Omron CX-Programmer project NewProject (CX-Programmer 9.75)

# PLC NewPLC1: CP2E-N N

## Program NewProgram1 (cyclic task 0)

### Section Section1

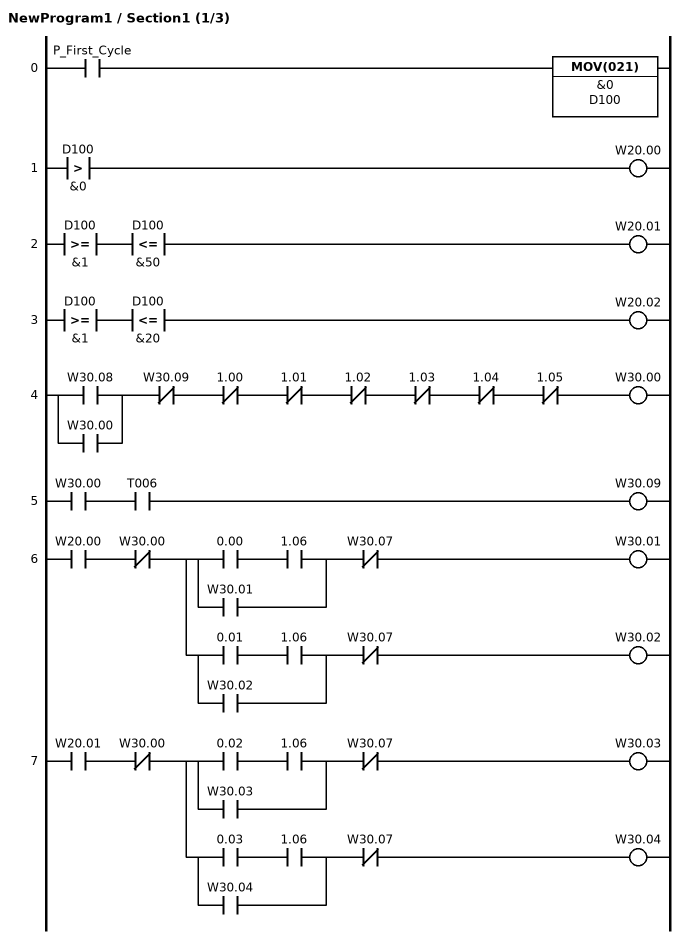
; rung 0
LD P_First_Cycle
MOV(021) &0 D100
; rung 1
LD>(320) D100 &0
OUT W20.00
; rung 2
LD>=(325) D100 &1
AND<=(315) D100 &50
OUT W20.01
; rung 3
LD>=(325) D100 &1
AND<=(315) D100 &20
OUT W20.02
; rung 4
LD W30.08
OR W30.00
ANDNOT W30.09
ANDNOT 1.00
ANDNOT 1.01
ANDNOT 1.02
ANDNOT 1.03
ANDNOT 1.04
ANDNOT 1.05
OUT W30.00
; rung 5
LD W30.00
AND T006
OUT W30.09
; rung 6
LD W20.00
ANDNOT W30.00
OUT TR0
LD 0.00
AND 1.06
OR W30.01
ANDLD
ANDNOT W30.07
OUT W30.01
LD TR0
LD 0.01
AND 1.06
OR W30.02
ANDLD
ANDNOT W30.07
OUT W30.02
; rung 7
LD W20.01
ANDNOT W30.00
OUT TR0
LD 0.02
AND 1.06
OR W30.03
ANDLD
ANDNOT W30.07
OUT W30.03
LD TR0
LD 0.03
AND 1.06
OR W30.04
ANDLD
ANDNOT W30.07
OUT W30.04

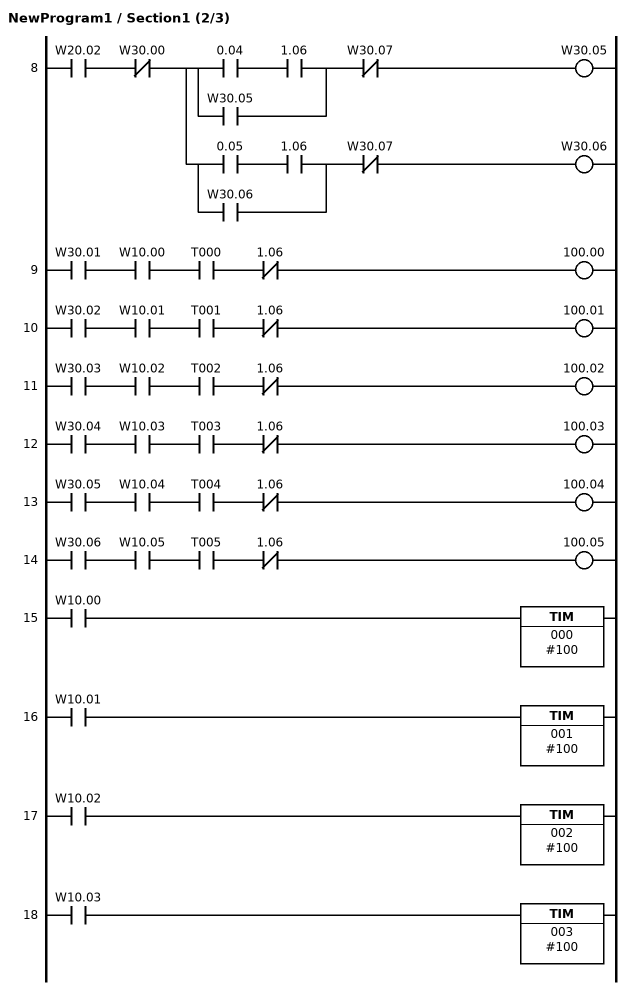
; rung 8
LD W20.02
ANDNOT W30.00
OUT TR0
LD 0.04
AND 1.06
OR W30.05
ANDLD
ANDNOT W30.07
OUT W30.05
LD TR0
LD 0.05
AND 1.06
OR W30.06
ANDLD
ANDNOT W30.07
OUT W30.06
; rung 9
LD W30.01
AND W10.00
AND T000
ANDNOT 1.06
OUT 100.00
; rung 10
LD W30.02
AND W10.01
AND T001
ANDNOT 1.06
OUT 100.01
; rung 11
LD W30.03
AND W10.02
AND T002
ANDNOT 1.06
OUT 100.02
; rung 12
LD W30.04
AND W10.03
AND T003
ANDNOT 1.06
OUT 100.03
; rung 13
LD W30.05
AND W10.04
AND T004
ANDNOT 1.06
OUT 100.04
; rung 14
LD W30.06
AND W10.05
AND T005
ANDNOT 1.06
OUT 100.05
; rung 15
LD W10.00
TIM 000 #100
; rung 16
LD W10.01
TIM 001 #100
; rung 17
LD W10.02
TIM 002 #100
; rung 18
LD W10.03
TIM 003 #100

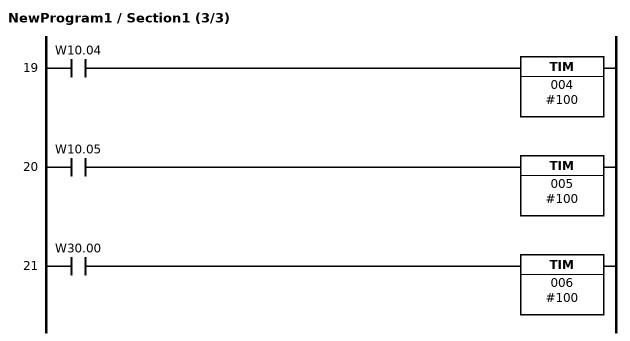
; rung 19
LD W10.04
TIM 004 #100
; rung 20
LD W10.05
TIM 005 #100
; rung 21
LD W30.00
TIM 006 #100

### Section END
; rung 0
END(001)